// TIA Portal V20 export
TYPE "LConSMC_typeTorquePrecontrolConfig"
// Konfiguration des Technologiereglers (Tänzer oder Zugmessdose) / Configuration parameters for technology controller (Dancer or load cell)
// stored: Access Published
   STRUCT
      useSetValForFrictionComp : Bool := FALSE;   // TRUE: Drehzahl-Sollwert wird für die Kompensastion der Reibung verwendet FALSE: Drehzahl-Istwert wird für die Kompensation der Reibung verwendet / TRUE: Use speed setpoint for friction compensation FALSE: Use speed actual value
      frictionAdjustment : Real := 0.0;   // Multiplikativer Faktor zur Adaption des Reibmomentes (1.0 = 100%) / Multiplicative adaption factor for friction torque (1.0 = 100%)
      xn_speedValues { S7_SetPoint := 'True'} : "LConSMC_typeBreakPointTable";   // [1/min] Drehzahlwerte der Reibkennlinie / [1/min] Speed values for fiction characteristic
      yn_torqueValues { S7_SetPoint := 'True'} : "LConSMC_typeBreakPointTable";   // [Nm oder lbf ft] Drehmomentenwerte der Reibkennlinie / [Nm or lbf ft] Torque values for friction characteristic
      sizeOfArray : Int := 20;   // Anzahl verwendeter Stützpunkte der Reibkennlinie / Size of friction characteristic array
      loadGear { S7_SetPoint := 'True'} : "LConSMC_typeLoadGear";   // Motorgetriebe / Load gear settings
      MaterialWidth : LReal := 0.0;   // [m or inch] Materialbreite / [m or inch] Width of the web
      MaterialDensity : LReal := 0.0;   // [kg/m^3 oder lb / ft^3 ] Materialdichte / [kg/m^3 or lb / ft^3 ] Material density
      MaterialFillFactor : Real := 1.0;   // Materialfüllfaktor (1.0 = 100%) Skallierungsfaktor für die Berechnung der Materialträgheit (wenn beispeilsweise kein Vollmaterial gewickelt wird) / Material fill factor (1.0-100%) Scaling factor for calculation of the material intertia (e.g. no solid material is winded)
      JFixed : LReal;   // [kgm^2] / [lbft^2] Trägheit bezogen auf Motorseite (ohne Motor, z.B. Getriebe) / [kgm^2] / [lbft^2] Inertia on drive side (without drive, e.g. gear box)
      JMandrel : LReal;   // [kgm^2] / [lbft^2] Trägheit auf der Lastseite (z.B. Rolle) / [kgm^2] / [lbft^2] Inertia on load side (e.g. mandrel)
      JMotor : LReal;   // [kgm^2] / [lbft^2] Motorträgheit / [kgm^2] / [lbft^2] Drive inertia
      tensionAdjustment : Real := 0.0;   // Multiplikativer Faktor zur Adaption des Zugmomentes (1.0 = 100%) / Multiplicative adaption factor for tension torque (1.0 = 100%)
      accelerationAdjustment : Real := 1.0;   // Multiplikativer Faktor zur Adaption des Beschleunigungsmomentes aus der Bahnbeschleunigung (1.0 = 100%) / Multiplicative adaption factor for acceleration torque from web acceleration (1.0 = 100%)
      dDdTAdjustment : Real := 0.0;   // Multiplikativer Faktor zur Adaption des Beschleunigungsmomentes welches aus der Durchmesseränderung entsteht (1.0 = 100%) / Multiplicative adaption factor for acceleration torque based on diameter change (1.0 = 100%)
      upperTorqueLimit : LReal := 1.0;   // [%] 1.0 = 100% Obere Drehmomentengrenze 0-200% des Bezugsmomentes / [%] 1.0 = 100% Upper torque limit 0..200% of nominal torque
      lowerTorqueLimit : LReal := -1.0;   // [%] 1.0 = 100% Untere Drehmomentengrenze 0-200% des Bezugsmomentes / [%] 1.0 = 100% Lower torque limit (0..-200% of nominal torque)
      referenceTorque : LReal;   // Referenzdrehmoment (SINAMICS p2003) !Nur notwendig wenn "getAxisConfigAtStart" = FALSE! / Reference torque (SINAMICS p2003) !Only necessary if "getAxisConfigAtStart" = FALSE!
      additiveTorque : LReal := 0.0;   // [Nm oder Lbf ft] Additives Zusatzmoment auf Motorseite für Aufwickler (z.B. zur Kompensation des Losbrechmomentes). Das Moment wirkt in Aufwickelrichtung und ist nur für "typeOfWinder" = 0/1 / [Nm or Lbf ft] Additive torque value on drive side for rewinder (.e.g. compensation of breakawy torque). The torque is in rewinding directio and only active of "typeOfWinder" = 0/1
   END_STRUCT;
   // xn_speedValues.values[0..19] := 0.0;
   // yn_torqueValues.values[0..19] := 0.0;
END_TYPE
